TYPE ST_DBResult :
STRUCT
	strCode : STRING(150);
	nExpiryStatus : DINT;
	(*nNumberOfchildren : INT;*)

(* nExpiryStatus:
0 - Expired
1 - Unknown - probaly due to reanimation. should still be successful
2 - Not Expired - OK*)
END_STRUCT
END_TYPE

(* stored: Version 1.1.0.1, ProductVersion 3.1.4024.15
   DUT ST_DBResult: Id {2ba63629-c2c1-40ba-9a0d-12fb56a5b11e} *)
